PROGRAM MAIN
VAR
END_VAR

END_PROGRAM

(* stored: Version 1.1.0.1
   POU MAIN: Id {61422c51-83de-45d6-9242-5ca335c20301} *)
